Fanuc KAREL source: KO00138.KL

PROGRAM KO00138
%NOLOCKGROUP
VAR
  R: REAL
  CFG: CONFIG
  OUT: XYZWPR
  N: REAL
BEGIN
  N = 1
  R = 2.0
  CFG.CFG_FLIP = TRUE
  OUT = POS(R, R, N, R, R, R, CFG)
END KO00138
